TYPE ST_Coordinates :
STRUCT
	HEIGHT : LREAL;
	DISTANCE : LREAL;
END_STRUCT
END_TYPE

(* stored: Version 1.1.0.1, ProductVersion 3.1.4026.12
   DUT ST_Coordinates: Id {eed01825-6221-49ba-8bb7-049462cb1d1a} *)
